	    // Manage step transitions and reset
	    #_step(forceReset := NOT #activate,
	           step := #step);
	    #_stepTracker.actual := #step.actual;
	END_REGION

	REGION Equipment Modules
	    REGION Vacuum: Commands
	        CASE #step.actual OF
	            VacHop_FlowThrough_Steps#RESET_STEP:
	                // Set vacuum to idle
	                #cmd_em_vacuum := _.EM_Vac.Vac_Cmd#IDLE;

	            VacHop_FlowThrough_Steps#INITIAL:
	                // Start vacuum or wait for idle
	                IF #em_vacuum_startVacuum_idle THEN
	                    #cmd_em_vacuum := _.EM_Vac.Vac_Cmd#IDLE;
	                ELSE
	                    #cmd_em_vacuum := _.EM_Vac.Vac_Cmd#START_VACUUM;
	                END_IF;
	            ELSE
	                // Maintain vacuum active
	                #cmd_em_vacuum := _.EM_Vac.Vac_Cmd#START_VACUUM;
	        END_CASE;

	    END_REGION

	    REGION Outlet Valve: Command
	        CASE #step.actual OF
	            VacHop_FlowThrough_Steps#RESET_STEP:
	                // Set outlet valve to idle
	                #cmd_em_outVlv := _.EM_outVlv.OutVlv_Cmd#IDLE;

	            VacHop_FlowThrough_Steps#INITIAL..VacHop_FlowThrough_Steps#CREATE_VACUUM:
	                // Open outlet valve or wait for close
	                IF NOT #em_outVlv_outletClose THEN
	                    #cmd_em_outVlv := _.EM_outVlv.OutVlv_Cmd#OPEN_OUTLET;

	                END_IF;
	            ELSE
	                // Maintain outlet valve open
	                #cmd_em_outVlv := _.EM_outVlv.OutVlv_Cmd#OPEN_OUTLET;

	        END_CASE;

	    END_REGION

	END_REGION

	REGION Control Modules: Commands
	    //********************************************************
	    // NA
	    //********************************************************

	END_REGION

	REGION Feedbacks
	    // na

	END_REGION

	REGION Status
	    // System idle when not activated
	    #status.idle := NOT #activate;

	    // System done when flowthrough complete
	    #status.done := NOT #status.idle AND #cm_inPosition AND #em_idleOrDone AND (#step.actual = VacHop_FlowThrough_Steps#READY);

	    //System busy during flowthrough sequence
	    #status.busy := NOT #status.idle AND NOT #status.done;

	END_REGION


END_FUNCTION_BLOCK
END_NAMESPACE

NAMESPACE EM_VacHop
TYPE VacHop_interface
{ Published := 'TRUE' }
VERSION : 0.1
   STRUCT
      cmd { ExternalAccessible := 'False'; ExternalVisible := 'False'; ExternalWritable := 'False'} : VacHop_Cmd;
      status { ExternalAccessible := 'False'; ExternalVisible := 'False'; ExternalWritable := 'False'; S7_SetPoint := 'False'} : _.LIB.Util_status;
      modesStatus { ExternalAccessible := 'False'; ExternalVisible := 'False'; ExternalWritable := 'False'; S7_SetPoint := 'False'} : VacHop_interface_modesStatus;
      feedbacks { ExternalAccessible := 'False'; ExternalVisible := 'False'; ExternalWritable := 'False'; S7_SetPoint := 'False'} : VacHop_interface_feedbacks;
   END_STRUCT;

END_TYPE
END_NAMESPACE

NAMESPACE EM_VacHop
FUNCTION_BLOCK EM_VacHop_evacuate
{ S7_Optimized_Access := 'TRUE' ; Published := 'TRUE' }
VERSION : 0.1
   VAR_INPUT
      enableStepTransition { ExternalAccessible := 'False'; ExternalVisible := 'False'; ExternalWritable := 'False'} : Bool := true;   // Enable Step Transition
      parameters { ExternalAccessible := 'False'; ExternalVisible := 'False'; ExternalWritable := 'False'} : VacHop_Evacuate_Params;
      activate { ExternalAccessible := 'False'; ExternalVisible := 'False'; ExternalWritable := 'False'} : Bool;
      cm_inPosition { ExternalAccessible := 'False'; ExternalVisible := 'False'; ExternalWritable := 'False'} : Bool;   // CM in position
      em_idleOrDone { ExternalAccessible := 'False'; ExternalVisible := 'False'; ExternalWritable := 'False'} : Bool;   // EM Idle or Done
      em_vacuum_startVacuum_idle { ExternalAccessible := 'False'; ExternalVisible := 'False'; ExternalWritable := 'False'} : Bool;   // EM Vacuum: Start Vacuum mode idle
      em_outVlv_outletClose { ExternalAccessible := 'False'; ExternalVisible := 'False'; ExternalWritable := 'False'} : Bool;   // EM_OutVlv: outlet valve is open
   END_VAR

   VAR_OUTPUT
      cmd_em_vacuum { ExternalAccessible := 'False'; ExternalVisible := 'False'; ExternalWritable := 'False'} : _.EM_Vac.Vac_Cmd;   // EM_Vacuum: Command
      cmd_em_outVlv { ExternalAccessible := 'False'; ExternalVisible := 'False'; ExternalWritable := 'False'} : _.EM_OutVlv.OutVlv_Cmd;   // EM_OutVlv: Command
   END_VAR

   VAR
      status { ExternalAccessible := 'False'; ExternalVisible := 'False'; ExternalWritable := 'False'; S7_SetPoint := 'False'} : _.LIB.Util_modeStatus;   // Mode status
      feedbacks { ExternalAccessible := 'False'; ExternalVisible := 'False'; ExternalWritable := 'False'; S7_SetPoint := 'False'} : VacHop_Evacuate_Feedbacks;   // Feedbacks
      step { ExternalAccessible := 'False'; ExternalVisible := 'False'; ExternalWritable := 'False'; S7_SetPoint := 'False'} : _.LIB.Util_Step;   // Step status
      _step { ExternalAccessible := 'False'; ExternalVisible := 'False'; ExternalWritable := 'False'; S7_SetPoint := 'False'} : _.LIB.Step;   // Step instance
      _stepTracker { ExternalAccessible := 'False'; ExternalVisible := 'False'; ExternalWritable := 'False'} : Struct
         actual { ExternalAccessible := 'False'; ExternalVisible := 'False'; ExternalWritable := 'False'} : VacHop_Evacuate_Steps;   // Current step
         next { ExternalAccessible := 'False'; ExternalVisible := 'False'; ExternalWritable := 'False'} : VacHop_Evacuate_Steps;   // Next step
      END_STRUCT;
   END_VAR


BEGIN
	REGION Header
	    //********************************************************
	    // EM_VacHop_evacuate Logic
	    // Description:
	    // - Manages the evacuation sequence for the vacuum hopper, closing the outlet and starting the vacuum system.
	    //********************************************************

	    REGION Revision History
	        (*
	        Author      Date        Change
	        GEA-VAR     2025-05-15  Initial version
	        *)
	    END_REGION
	END_REGION

	REGION Step
	    IF #activate THEN
	        CASE #step.actual OF
	                // Idle state, no sequence active
	            VacHop_Evacuate_Steps#INITIAL:
	                #_stepTracker.next := VacHop_Evacuate_Steps#CLOSE_OUTLET;

	                // Close outlet valve
	            VacHop_Evacuate_Steps#CLOSE_OUTLET:
	                #_stepTracker.next := VacHop_Evacuate_Steps#CREATE_VACUUM;

	                //  Start vacuum system
	            VacHop_Evacuate_Steps#CREATE_VACUUM:
	                #_stepTracker.next := VacHop_Evacuate_Steps#DONE;

	                //  Evacuation sequence complete
	            VacHop_Evacuate_Steps#DONE:
	                ;

	                // Handle invalid step
	            ELSE
	                // Reset to idle on invalid step
	                #step.actual := #_stepTracker.next := VacHop_Evacuate_Steps#INITIAL;
	        END_CASE;

	        // Advance step when module positioned
	        IF #enableStepTransition AND #cm_inPosition AND #em_idleOrDone THEN
	            #step.actual := #_stepTracker.next;
	        END_IF;

	    END_IF;

	    // Manage step transitions and reset
	    #_step(forceReset := NOT #activate,
	           step := #step);
	    #_stepTracker.actual := #step.actual;

	END_REGION

	REGION Equipment Modules
	    REGION Vacuum: Commands
	        CASE #step.actual OF
	            VacHop_Evacuate_Steps#RESET_STEP:
	                #cmd_em_vacuum := _.EM_Vac.Vac_Cmd#IDLE;

	            VacHop_Evacuate_Steps#INITIAL..VacHop_Evacuate_Steps#CLOSE_OUTLET:
	                IF #em_vacuum_startVacuum_idle THEN
	                    #cmd_em_vacuum := _.EM_Vac.Vac_Cmd#IDLE;
	                ELSE
	                    #cmd_em_vacuum := _.EM_Vac.Vac_Cmd#START_VACUUM;
	                END_IF;
	            ELSE
	                #cmd_em_vacuum := _.EM_Vac.Vac_Cmd#START_VACUUM;
	        END_CASE;

	    END_REGION

	    REGION Outlet Valve: Command
	        CASE #step.actual OF
	            VacHop_Evacuate_Steps#INITIAL..VacHop_Evacuate_Steps#CLOSE_OUTLET:
	                IF NOT #em_outVlv_outletClose THEN
	                    #cmd_em_outVlv := _.EM_outVlv.OutVlv_Cmd#CLOSE_OUTLET;
	                ELSE
	                    #cmd_em_outVlv := _.EM_outVlv.OutVlv_Cmd#IDLE;
	                END_IF;
	            ELSE
	                #cmd_em_outVlv := _.EM_outVlv.OutVlv_Cmd#IDLE;

	        END_CASE;

	    END_REGION

	END_REGION

	REGION Control Modules: Commands
	    //********************************************************
	    // NA
	    //********************************************************

	END_REGION

	REGION Feedbacks
	    // NA

	END_REGION

	REGION Status
	    // System idle when not activated
	    #status.idle := NOT #activate;

	    // System done when evacuation complete
	    #status.done := NOT #status.idle AND #cm_inPosition AND #em_idleOrDone AND (#step.actual = VacHop_Evacuate_Steps#DONE);

	    // System busy during evacuation sequence
	    #status.busy := NOT #status.idle AND NOT #status.done;

	END_REGION


END_FUNCTION_BLOCK
END_NAMESPACE

NAMESPACE EM_VacHop
FUNCTION_BLOCK EM_VacHop_openHopper
{ S7_Optimized_Access := 'TRUE' ; Published := 'TRUE' }
VERSION : 0.1
   VAR_INPUT
      enableStepTransition { ExternalAccessible := 'False'; ExternalVisible := 'False'; ExternalWritable := 'False'} : Bool := true;   // Enable Step Transition
      parameters { ExternalAccessible := 'False'; ExternalVisible := 'False'; ExternalWritable := 'False'} : VacHop_OpenHopper_Params;   // Open hopper parameters
      activate { ExternalAccessible := 'False'; ExternalVisible := 'False'; ExternalWritable := 'False'} : Bool;   // Activate open sequence
      cm_inPosition { ExternalAccessible := 'False'; ExternalVisible := 'False'; ExternalWritable := 'False'} : Bool;   // CM in position
      em_idleOrDone { ExternalAccessible := 'False'; ExternalVisible := 'False'; ExternalWritable := 'False'} : Bool;   // EM Idle or Done
      em_vacuum_idle { ExternalAccessible := 'False'; ExternalVisible := 'False'; ExternalWritable := 'False'} : Bool;   // EM Vacuum:  idle
      em_outVlv_outletClose { ExternalAccessible := 'False'; ExternalVisible := 'False'; ExternalWritable := 'False'} : Bool;   // EM_OutVlv outlet valve closed
   END_VAR

   VAR_OUTPUT
      cmd_em_vacuum { ExternalAccessible := 'False'; ExternalVisible := 'False'; ExternalWritable := 'False'} : _.EM_Vac.Vac_Cmd;   // EM_Vacuum: Command
      cmd_em_outVlv { ExternalAccessible := 'False'; ExternalVisible := 'False'; ExternalWritable := 'False'} : _.EM_OutVlv.OutVlv_Cmd;   // EM_Hopper: Command
   END_VAR

   VAR
      status { ExternalAccessible := 'False'; ExternalVisible := 'False'; ExternalWritable := 'False'; S7_SetPoint := 'False'} : _.LIB.Util_modeStatus;   // Mode status
      feedbacks { ExternalAccessible := 'False'; ExternalVisible := 'False'; ExternalWritable := 'False'; S7_SetPoint := 'False'} : VacHop_OpenHopper_Feedbacks;   // Feedbacks
      step { ExternalAccessible := 'False'; ExternalVisible := 'False'; ExternalWritable := 'False'; S7_SetPoint := 'False'} : _.LIB.Util_Step;   // Step status
      _step { ExternalAccessible := 'False'; ExternalVisible := 'False'; ExternalWritable := 'False'; S7_SetPoint := 'False'} : _.LIB.Step;   // Step instance
      _stepTracker { ExternalAccessible := 'False'; ExternalVisible := 'False'; ExternalWritable := 'False'} : Struct
         actual { ExternalAccessible := 'False'; ExternalVisible := 'False'; ExternalWritable := 'False'} : VacHop_OpenHopper_Steps;   // Current step
         next { ExternalAccessible := 'False'; ExternalVisible := 'False'; ExternalWritable := 'False'} : VacHop_OpenHopper_Steps;   // Next step
      END_STRUCT;
   END_VAR


BEGIN
	REGION Header
	    //********************************************************
	    // EM_VacHop_openHopper Logic
	    // Description:
	    // - Manages the hopper outlet opening sequence for the vacuum hopper, stopping vacuum and opening the outlet valve.
	    //********************************************************

	    REGION Revision History
	        (*
	        Author      Date        Change
	        GEA-VAR     2025-05-15  Initial version
	        *)
	    END_REGION
	END_REGION

	REGION Step
	    IF #activate THEN
	        CASE #step.actual OF
	                // Idle state, no sequence active
	            VacHop_OpenHopper_Steps#INITIAL:
	                #_stepTracker.next := VacHop_OpenHopper_Steps#STOP_VACUUM;

	                // Stop vacuum system
	            VacHop_OpenHopper_Steps#STOP_VACUUM:
	                #_stepTracker.next := VacHop_OpenHopper_Steps#OPEN_OUTLET;

	                //  Open outlet valve
	            VacHop_OpenHopper_Steps#OPEN_OUTLET:
	                #_stepTracker.next := VacHop_OpenHopper_Steps#DONE;

	                //  Outlet valve opened, sequence complete
	            VacHop_OpenHopper_Steps#DONE:
	                ;

	                // Handle invalid step
	            ELSE
	                // Reset to idle on invalid step
	                #step.actual := #_stepTracker.next := VacHop_OpenHopper_Steps#INITIAL;
	        END_CASE;

	        // Advance step when module positioned
	        IF #enableStepTransition AND #cm_inPosition AND #em_idleOrDone THEN
	            #step.actual := #_stepTracker.next;
	        END_IF;

	    END_IF;

	    // Manage step transitions and reset
	    #_step(forceReset := NOT #activate,
	           step := #step);
	    #_stepTracker.actual := #step.actual;

	END_REGION

	REGION Control/Equipment Modules and Modes: Commands

	    REGION Vacuum: Commands
	        CASE #step.actual OF
	            VacHop_OpenHopper_Steps#INITIAL..VacHop_OpenHopper_Steps#STOP_VACUUM:
	                IF #em_vacuum_idle THEN
	                    #cmd_em_vacuum := _.EM_Vac.Vac_Cmd#IDLE;
	                ELSE
	                    #cmd_em_vacuum := _.EM_Vac.Vac_Cmd#STOP_VACUUM;
	                END_IF;
	            ELSE
	                #cmd_em_vacuum := _.EM_Vac.Vac_Cmd#IDLE;
	        END_CASE;

	    END_REGION

	    REGION Outlet Valve: Command
	        CASE #step.actual OF
	            VacHop_OpenHopper_Steps#RESET_STEP:
	                #cmd_em_outVlv := _.EM_outVlv.OutVlv_Cmd#IDLE;

	            VacHop_OpenHopper_Steps#INITIAL..VacHop_OpenHopper_Steps#STOP_VACUUM:
	                IF NOT #em_outVlv_outletClose THEN
	                    #cmd_em_outVlv := _.EM_outVlv.OutVlv_Cmd#OPEN_OUTLET;
	                ELSE
	                    #cmd_em_outVlv := _.EM_outVlv.OutVlv_Cmd#IDLE;
	                END_IF;
	            ELSE
	                #cmd_em_outVlv := _.EM_outVlv.OutVlv_Cmd#OPEN_OUTLET;
	        END_CASE;

	    END_REGION

	END_REGION

	REGION Control Modules: Commands
	    //********************************************************
	    // NA
	    //********************************************************

	END_REGION

	REGION Feedbacks
	    // NA

	END_REGION

	REGION Status
	    // System idle when not activated
	    #status.idle := NOT #activate;

	    // System done when hopper opened
	    #status.done := (NOT #status.idle) AND #cm_inPosition AND #em_idleOrDone AND (#step.actual = VacHop_OpenHopper_Steps#DONE);

	    // System busy during open sequence
	    #status.busy := NOT #status.idle AND NOT #status.done;

	END_REGION


END_FUNCTION_BLOCK
END_NAMESPACE

NAMESPACE EM_VacHop
FUNCTION_BLOCK EM_VacHop_vent
{ S7_Optimized_Access := 'TRUE' ; Published := 'TRUE' }
VERSION : 0.1
   VAR_INPUT
      enableStepTransition { ExternalAccessible := 'False'; ExternalVisible := 'False'; ExternalWritable := 'False'} : Bool := true;   // Enable Step Transition
      parameters { ExternalAccessible := 'False'; ExternalVisible := 'False'; ExternalWritable := 'False'} : VacHop_Vent_Params;   // Vent parameters
      activate { ExternalAccessible := 'False'; ExternalVisible := 'False'; ExternalWritable := 'False'} : Bool;   // Activate vent sequence
      cm_inPosition { ExternalAccessible := 'False'; ExternalVisible := 'False'; ExternalWritable := 'False'} : Bool;   // CM in position
      em_idleOrDone { ExternalAccessible := 'False'; ExternalVisible := 'False'; ExternalWritable := 'False'} : Bool;   // EM Idle or Done
      em_vacuum_idle { ExternalAccessible := 'False'; ExternalVisible := 'False'; ExternalWritable := 'False'} : Bool;   // EM Vacuum:  idle
      em_outVlv_outletClose { ExternalAccessible := 'False'; ExternalVisible := 'False'; ExternalWritable := 'False'} : Bool;   // EM_outVlv: outlet valve is closed
   END_VAR

   VAR_OUTPUT
      cmd_em_vacuum { ExternalAccessible := 'False'; ExternalVisible := 'False'; ExternalWritable := 'False'} : _.EM_Vac.Vac_Cmd;   // EM_Vacuum: Command
      cmd_em_outVlv { ExternalAccessible := 'False'; ExternalVisible := 'False'; ExternalWritable := 'False'} : _.EM_OutVlv.OutVlv_Cmd;   // EM_outVlv: Command
      cmd_ventVlvOpen { ExternalAccessible := 'False'; ExternalVisible := 'False'; ExternalWritable := 'False'} : Bool;   // Command vent valve open
   END_VAR

   VAR
      status { ExternalAccessible := 'False'; ExternalVisible := 'False'; ExternalWritable := 'False'; S7_SetPoint := 'False'} : _.LIB.Util_modeStatus;   // Mode status
      feedbacks { ExternalAccessible := 'False'; ExternalVisible := 'False'; ExternalWritable := 'False'; S7_SetPoint := 'False'} : VacHop_Vent_Feedbacks;   // Feedbacks
      step { ExternalAccessible := 'False'; ExternalVisible := 'False'; ExternalWritable := 'False'; S7_SetPoint := 'False'} : _.LIB.Util_Step;   // Step status
      _step { ExternalAccessible := 'False'; ExternalVisible := 'False'; ExternalWritable := 'False'; S7_SetPoint := 'False'} : _.LIB.Step;   // Step instance
      _stepTracker { ExternalAccessible := 'False'; ExternalVisible := 'False'; ExternalWritable := 'False'} : Struct
         actual { ExternalAccessible := 'False'; ExternalVisible := 'False'; ExternalWritable := 'False'} : VacHop_Vent_Steps;   // Current step
         next { ExternalAccessible := 'False'; ExternalVisible := 'False'; ExternalWritable := 'False'} : VacHop_Vent_Steps;   // Next step
      END_STRUCT;
   END_VAR


BEGIN
	REGION Header
	    //********************************************************
	    // EM_VacHop_vent Logic
	    // Description:
	    // - Manages the vent sequence for the vacuum hopper, stopping vacuum, closing outlet, and cycling the vent valve.
	    //********************************************************

	    REGION Revision History
	        (*
	        Author      Date        Change
	        GEA-VAR     2025-05-15  Initial version
	        *)
	    END_REGION
	END_REGION

	REGION Step
	    IF #activate THEN
	        CASE #step.actual OF
	                // Idle state, no sequence active
	            VacHop_Vent_Steps#INITIAL:
	                #_stepTracker.next := VacHop_Vent_Steps#STOP_VACUUM_AND_CLOSE_OUTLET;

	                // Stop vacuum and close outlet valve
	            VacHop_Vent_Steps#STOP_VACUUM_AND_CLOSE_OUTLET:
	                #_stepTracker.next := VacHop_Vent_Steps#OPEN_VENT_VALVE;

	                //  Open vent valve
	            VacHop_Vent_Steps#OPEN_VENT_VALVE:
	                #_stepTracker.next := VacHop_Vent_Steps#VENT_DELAY_ACTIVE;

	                //  Delay for venting
	            VacHop_Vent_Steps#VENT_DELAY_ACTIVE:
	                IF _.LIB.IsTimerExceeded(actualTimer:=#step.actualTimer, limit:=#parameters.ventTime) THEN
	                    #_stepTracker.next := VacHop_Vent_Steps#CLOSE_VENT_VALVE;
	                END_IF;

	                // Close vent valve
	            VacHop_Vent_Steps#CLOSE_VENT_VALVE:
	                #_stepTracker.next := VacHop_Vent_Steps#DONE;

	                // Vent sequence complete
	            VacHop_Vent_Steps#DONE:
	                ;

	                // Handle invalid step
	            ELSE
	                // Reset to idle on invalid step
	                #step.actual := #_stepTracker.next := VacHop_Vent_Steps#INITIAL;
	        END_CASE;

	        // Advance step when module positioned
	        IF #enableStepTransition AND #cm_inPosition AND #em_idleOrDone THEN
	            #step.actual := #_stepTracker.next;
	        END_IF;

	    END_IF;

	    // Manage step transitions and reset
	    #_step(forceReset:=NOT #activate,
	           step := #step);
	    #_stepTracker.actual := #step.actual;
	END_REGION

	REGION Actions
	    // NA

	END_REGION

	REGION Control/Equipment Modules and Modes: Commands
	    REGION Vacuum: Commands
	        CASE #step.actual OF
	            VacHop_Vent_Steps#INITIAL..VacHop_Vent_Steps#STOP_VACUUM_AND_CLOSE_OUTLET:
	                IF #em_vacuum_idle THEN
	                    #cmd_em_vacuum := _.EM_Vac.Vac_Cmd#IDLE;
	                ELSE
	                    #cmd_em_vacuum := _.EM_Vac.Vac_Cmd#STOP_VACUUM;
	                END_IF;
	            ELSE
	                #cmd_em_vacuum := _.EM_Vac.Vac_Cmd#IDLE;
	        END_CASE;

	    END_REGION

	    REGION Vacuum valve: Command
	        CASE #step.actual OF
	            VacHop_Vent_Steps#INITIAL..VacHop_Vent_Steps#STOP_VACUUM_AND_CLOSE_OUTLET:
	                IF NOT #em_outVlv_outletClose THEN
	                    #cmd_em_outVlv := _.EM_outVlv.OutVlv_Cmd#CLOSE_OUTLET;
	                ELSE
	                    #cmd_em_outVlv := _.EM_outVlv.OutVlv_Cmd#IDLE;
	                END_IF;
	            ELSE
	                #cmd_em_outVlv := _.EM_outVlv.OutVlv_Cmd#IDLE;
	        END_CASE;

	    END_REGION

	END_REGION

	REGION Control Modules: Commands
	    //********************************************************
	    // Vent Valve
	    //********************************************************
	    #cmd_ventVlvOpen := #activate AND (NOT (#step.actual = VacHop_Vent_Steps#CLOSE_VENT_VALVE)) AND (NOT ((#step.actual = VacHop_Vent_Steps#DONE)));


	END_REGION

	REGION #feedbacks
	    // Update feedback statuses
	    #feedbacks.venting := (#step.actual = VacHop_Vent_Steps#OPEN_VENT_VALVE) OR (#step.actual = VacHop_Vent_Steps#VENT_DELAY_ACTIVE);

	END_REGION

	REGION Status
	    // System idle when not activated
	    #status.idle := NOT #activate;

	    // System done when vent complete
	    #status.done := (NOT #status.idle) AND #cm_inPosition AND #em_idleOrDone AND (#step.actual = VacHop_Vent_Steps#DONE);

	    // System busy during vent sequence
	    #status.busy := NOT #status.idle AND NOT #status.done;

	END_REGION


END_FUNCTION_BLOCK
END_NAMESPACE

NAMESPACE EM_OutVlv
FUNCTION_BLOCK EM_OutVlv
{ S7_Optimized_Access := 'TRUE' ; Published := 'TRUE' }
VERSION : 0.1
   VAR_INPUT
      enableStepTransition { ExternalAccessible := 'False'; ExternalVisible := 'False'; ExternalWritable := 'False'} : Bool := True;   // Enable step transition
      outletValveInputs { ExternalAccessible := 'False'; ExternalVisible := 'False'; ExternalWritable := 'False'} : OutVlv_inputs;   // EM inputs
   END_VAR

   VAR_OUTPUT
      cm_inPosition { ExternalAccessible := 'False'; ExternalVisible := 'False'; ExternalWritable := 'False'} : Bool;   // CM in position
      cmd_outletVlvOpen { ExternalAccessible := 'False'; ExternalVisible := 'False'; ExternalWritable := 'False'} : Bool;   // Command: outlet valve open
   END_VAR

   VAR
      interface { ExternalAccessible := 'False'; ExternalVisible := 'False'; ExternalWritable := 'False'; S7_SetPoint := 'False'} : OutVlv_interface;
      parameters : OutVlv_parameters;
      _initialize { ExternalAccessible := 'False'; ExternalVisible := 'False'; ExternalWritable := 'False'; S7_SetPoint := 'False'} : EM_OutVlv_initialize;
      _purge { ExternalAccessible := 'False'; ExternalVisible := 'False'; ExternalWritable := 'False'; S7_SetPoint := 'False'} : EM_OutVlv_purge;
      _discharge { ExternalAccessible := 'False'; ExternalVisible := 'False'; ExternalWritable := 'False'; S7_SetPoint := 'False'} : EM_OutVlv_discharge;
      _holdPosition { ExternalAccessible := 'False'; ExternalVisible := 'False'; ExternalWritable := 'False'; S7_SetPoint := 'False'} : EM_OutVlv_holdPosition;
      _openOutlet { ExternalAccessible := 'False'; ExternalVisible := 'False'; ExternalWritable := 'False'; S7_SetPoint := 'False'} : EM_OutVlv_openOutlet;
      _closeOutlet { ExternalAccessible := 'False'; ExternalVisible := 'False'; ExternalWritable := 'False'; S7_SetPoint := 'False'} : EM_OutVlv_closeOutlet;
      _outputs { ExternalAccessible := 'False'; ExternalVisible := 'False'; ExternalWritable := 'False'} : Struct
         cmd_outletVlvOpen { ExternalAccessible := 'False'; ExternalVisible := 'False'; ExternalWritable := 'False'} : Bool;
      END_STRUCT;
   END_VAR

   VAR_TEMP
      temp_mode_idle_or_done : Bool;
   END_VAR


BEGIN
	REGION Header
	    //********************************************************
	    // EM_OutVlv Logic
	    // Description:
	    // - Main controller for the outlet valvce system.
	    //********************************************************

	    REGION Revision History
	        (*
	            Author      Date        Change
	            GEA-VAR     15MAY25     Initial version
	        *)
	    END_REGION

	END_REGION

	REGION Check CM/EM(mode) in position
	    // Set control module position status
	    #cm_inPosition :=
	        (#_outputs.cmd_outletVlvOpen AND #outletValveInputs.outletVlv_isOpen) OR
	        ((NOT #_outputs.cmd_outletVlvOpen) AND #outletValveInputs.outletVlv_isClosed);

	    #temp_mode_idle_or_done :=
	        (#_openOutlet.status.idle OR #_openOutlet.status.done) AND
	        (#_closeOutlet.status.idle OR #_closeOutlet.status.done);

	END_REGION

	REGION Initialize
	    // Run initialization sequence
	    #_initialize(enableStepTransition:=#enableStepTransition,
	                 activate:=(#interface.cmd = OutVlv_Cmd#INITIALIZE),
	                 cm_inPosition:=#cm_inPosition,
	                 mode_idleOrDone:=#temp_mode_idle_or_done);

	END_REGION

	REGION Purge
	    REGION Parameters
	        // Configure parameters for the purge count
	        #_purge.parameters.startDelay := #parameters.fixed.purgeStartDelay;
	        #_purge.parameters.count := #parameters.fixed.purgeCount;
	        #_purge.parameters.outletVlvOpenDelay := #parameters.fixed.purgeOutletVlvOpenDelay;
	        #_purge.parameters.outletVlvCloseDelay := #parameters.fixed.purgeOutletVlvCloseDelay;

	    END_REGION

	    // Activate Purge sequence on command
	    #_purge(enableStepTransition:=#enableStepTransition,
	            activate := (#interface.cmd = OutVlv_Cmd#PURGE),
	            cm_inPosition:=#cm_inPosition,
	            mode_idleOrDone:=#temp_mode_idle_or_done,
	            outletVlv_isOpen:=#outletValveInputs.outletVlv_isOpen);
	END_REGION

	REGION Discharge
	    // Configure parameters for the discharge mode
	    REGION Parameters
	        #_discharge.parameters.dischargeTime := #parameters.variable.dischargeTime;

	    END_REGION

	    // Activate Purge sequence on command
	    #_discharge(enableStepTransition:=#enableStepTransition,
	                activate := (#interface.cmd = OutVlv_Cmd#DISCHARGE),
	                cm_inPosition:=#cm_inPosition,
	                mode_idleOrDone:=#temp_mode_idle_or_done);
	END_REGION

	REGION Hold Position
	    // Configure parameters for the Hold Position mode
	    REGION Parameters
	        #_holdPosition.parameters.na := FALSE;

	    END_REGION

	    // Activate Hold Position sequence on command
	    #_holdPosition(enableStepTransition:=#enableStepTransition,
	                   activate := (#interface.cmd = OutVlv_Cmd#HOLD_POSITION),
	                   cm_inPosition := #cm_inPosition,
	                   mode_idleOrDone := #temp_mode_idle_or_done,
	                   outletVlv_isClosed:=#outletValveInputs.outletVlv_isClosed);
	END_REGION

	REGION Open Outlet
	    // Configure parameters for the open outlet delay
	    REGION Parameters
	        IF #_purge.cmd_modeOpenOutlet THEN
	            #_openOutlet.parameters.vlvOpenDelay := #_purge.parameters.outletVlvOpenDelay;
	        ELSE
	            #_openOutlet.parameters.vlvOpenDelay := #parameters.fixed.outletVlvOpenDelay;
	        END_IF;

	    END_REGION

	    // Activate Open Outlet sequence when commanded or required by initialization, purge, discharge or holdPosition
	    #_openOutlet(enableStepTransition:=#enableStepTransition,
	                 activate := (#interface.cmd = OutVlv_Cmd#OPEN_OUTLET) OR #_initialize.cmd_modeOpenOutlet OR #_purge.cmd_modeOpenOutlet OR #_discharge.cmd_modeOpenOutlet OR #_holdPosition.cmd_modeOpenOutlet,
	                 cm_inPosition:=#cm_inPosition,
	                 outletVlv_isOpen:=#outletValveInputs.outletVlv_isOpen);

	END_REGION

	REGION Close Outlet
	    // Configure parameters for the close outlet delay
	    REGION Parameters
	        IF #_purge.cmd_modeCloseOutlet THEN
	            #_closeOutlet.parameters.vlvCloseDelay := #_purge.parameters.outletVlvCloseDelay;
	        ELSE
	            #_closeOutlet.parameters.vlvCloseDelay := #parameters.fixed.outletVlvCloseDelay;
	        END_IF;

	    END_REGION

	    // Activate Close Outlet sequence when commanded or required by initialization, purge, discharge or holdPosition
	    #_closeOutlet(enableStepTransition:=#enableStepTransition,
	                  activate := (#interface.cmd = OutVlv_Cmd#CLOSE_OUTLET) OR #_initialize.cmd_modeCloseOutlet OR #_purge.cmd_modeCloseOutlet OR #_discharge.cmd_modeCloseOutlet OR #_holdPosition.cmd_modeCloseOutlet,
	                  cm_inPosition:=#cm_inPosition,
	                  outletVlv_isOpen := #outletValveInputs.outletVlv_isOpen,
	                  outletVlv_isClosed := #outletValveInputs.outletVlv_isClosed);
	END_REGION


	REGION Outputs
	    // Combine valve commands from outlet sequences
	    #cmd_outletVlvOpen := #_outputs.cmd_outletVlvOpen := #_openOutlet.cmd_outletVlvOpen OR #_closeOutlet.cmd_outletVlvOpen;

	END_REGION

	REGION Feedbacks
	    // Update mode feedbacks
	    #interface.feedbacks.outletOpen := #outletValveInputs.outletVlv_isOpen;
	    #interface.feedbacks.openingOutlet := (NOT #outletValveInputs.outletVlv_isOpen) AND #cmd_outletVlvOpen;
	    #interface.feedbacks.outletClose := #outletValveInputs.outletVlv_isClosed;
	    #interface.feedbacks.closingOutlet := (NOT #outletValveInputs.outletVlv_isClosed) AND (#interface.cmd <> OutVlv_Cmd#IDLE) AND  (NOT #cmd_outletVlvOpen);
	    #interface.feedbacks.held := #_holdPosition.feedbacks.held;

	    REGION Modes
	        #interface.feedbacks.modes.initialize := #_initialize.feedbacks;
	        #interface.feedbacks.modes.openOutlet := #_openOutlet.feedbacks;
	        #interface.feedbacks.modes.closeOutlet := #_closeOutlet.feedbacks;
	        #interface.feedbacks.modes.purge := #_purge.feedbacks;
	        #interface.feedbacks.modes.discharge := #_discharge.feedbacks;
	        #interface.feedbacks.modes.holdPosition := #_holdPosition.feedbacks;

	    END_REGION

	END_REGION


	REGION Check CM/EM(mode) in position
	    // Set control module position status
	    #cm_inPosition :=
	        (#_outputs.cmd_outletVlvOpen AND #outletValveInputs.outletVlv_isOpen) OR
	        ((NOT #_outputs.cmd_outletVlvOpen) AND #outletValveInputs.outletVlv_isClosed);

	    // Check if modes are idle or done
	    #temp_mode_idle_or_done :=
	        (#_openOutlet.status.idle OR #_openOutlet.status.done) AND
	        (#_closeOutlet.status.idle OR #_closeOutlet.status.done);

	END_REGION

	REGION Status
	    #interface.status.done := #_initialize.status.done OR #_purge.status.done OR #_discharge.status.done OR #_holdPosition.status.done OR
	    ((NOT (#_initialize.status.busy OR #_purge.status.busy OR #_discharge.status.busy OR #_holdPosition.status.busy)) AND (#_openOutlet.status.done OR #_closeOutlet.status.done));
	    #interface.status.busy := #_initialize.status.busy OR #_openOutlet.status.busy OR #_closeOutlet.status.busy OR #_purge.status.busy OR #_discharge.status.busy;
	    #interface.status.idle := NOT (#interface.status.busy OR #interface.status.done);
	    #interface.status.stopAlmActive := _.EM.TODO.alm;
	    #interface.status.abortAlmActive := _.EM.TODO.alm;

	    // Modes
	    #interface.modesStatus.initialize := #_initialize.status;
	    #interface.modesStatus.openOutlet := #_openOutlet.status;
	    #interface.modesStatus.closeOutlet := #_closeOutlet.status;
	    #interface.modesStatus.purge := #_purge.status;
	    #interface.modesStatus.discharge := #_discharge.status;
	    #interface.modesStatus.holdPosition := #_holdPosition.status;

	END_REGION

END_FUNCTION_BLOCK
END_NAMESPACE

NAMESPACE EM_VacHop
FUNCTION_BLOCK EM_VacHop_discharge
{ S7_Optimized_Access := 'TRUE' ; Published := 'TRUE' }
VERSION : 0.1
   VAR_INPUT
      enableStepTransition { ExternalAccessible := 'False'; ExternalVisible := 'False'; ExternalWritable := 'False'} : Bool := true;   // Enable Step Transition
      parameters { ExternalAccessible := 'False'; ExternalVisible := 'False'; ExternalWritable := 'False'} : VacHop_Discharge_Params;   // Discharge parameters
      activate { ExternalAccessible := 'False'; ExternalVisible := 'False'; ExternalWritable := 'False'} : Bool;   // Activate discharge sequence
      cm_inPosition { ExternalAccessible := 'False'; ExternalVisible := 'False'; ExternalWritable := 'False'} : Bool;   // CM in position
      em_idleOrDone { ExternalAccessible := 'False'; ExternalVisible := 'False'; ExternalWritable := 'False'} : Bool;   // EM Idle or Done
      em_vacuum_idle { ExternalAccessible := 'False'; ExternalVisible := 'False'; ExternalWritable := 'False'} : Bool;   // EM vacuum idle
      em_outVlv_outletClose { ExternalAccessible := 'False'; ExternalVisible := 'False'; ExternalWritable := 'False'} : Bool;   // EM_OutVlv: outlet valve is closed
   END_VAR

   VAR_OUTPUT
      cmd_em_vacuum { ExternalAccessible := 'False'; ExternalVisible := 'False'; ExternalWritable := 'False'} : _.EM_Vac.Vac_Cmd;   // EM_Vac command
      cmd_em_outVlv { ExternalAccessible := 'False'; ExternalVisible := 'False'; ExternalWritable := 'False'} : _.EM_OutVlv.OutVlv_Cmd;   // EM_OutVlv command
   END_VAR

   VAR
      status { ExternalAccessible := 'False'; ExternalVisible := 'False'; ExternalWritable := 'False'; S7_SetPoint := 'False'} : _.LIB.Util_modeStatus;   // Mode status
      feedbacks { ExternalAccessible := 'False'; ExternalVisible := 'False'; ExternalWritable := 'False'; S7_SetPoint := 'False'} : VacHop_Discharge_Feedbacks;   // Feedbacks
      step { ExternalAccessible := 'False'; ExternalVisible := 'False'; ExternalWritable := 'False'; S7_SetPoint := 'False'} : _.LIB.Util_Step;   // Step status
      _step { ExternalAccessible := 'False'; ExternalVisible := 'False'; ExternalWritable := 'False'; S7_SetPoint := 'False'} : _.LIB.Step;   // Step instance
      _stepTracker { ExternalAccessible := 'False'; ExternalVisible := 'False'; ExternalWritable := 'False'} : Struct
         actual { ExternalAccessible := 'False'; ExternalVisible := 'False'; ExternalWritable := 'False'} : VacHop_Discharge_Steps;   // Current step
         next { ExternalAccessible := 'False'; ExternalVisible := 'False'; ExternalWritable := 'False'} : VacHop_Discharge_Steps;   // Next step
      END_STRUCT;
   END_VAR


BEGIN
	REGION Header
	    //********************************************************
	    // EM_VacHop_discharge Logic
	    // Description:
	    // - Manages the discharge sequence for the vacuum hopper, stopping vacuum and opening the outlet valve.
	    //********************************************************

	    REGION Revision History
	        (*
	        Author      Date        Change
	        GEA-VAR     2025-05-15  Initial version
	        *)
	    END_REGION
	END_REGION

	REGION Step
	    IF #activate THEN
	        CASE #step.actual OF
	                // Idle state, no sequence active
	            VacHop_Discharge_Steps#INITIAL:
	                #_stepTracker.next := VacHop_Discharge_Steps#STOP_VACUUM;

	                // Stop vacuum system
	            VacHop_Discharge_Steps#STOP_VACUUM:
	                #_stepTracker.next := VacHop_Discharge_Steps#DISCHARGE;

	                // Discharge product
	            VacHop_Discharge_Steps#DISCHARGE:
	                #_stepTracker.next := VacHop_Discharge_Steps#DONE;

	                // Discharge sequence complete
	            VacHop_Discharge_Steps#DONE:
	                ;

	                // Handle invalid step
	            ELSE
	                // Reset to idle on invalid step
	                #step.actual := #_stepTracker.next := VacHop_Discharge_Steps#INITIAL;
	        END_CASE;

	        // Advance step when module positioned
	        IF #enableStepTransition AND  #cm_inPosition AND #em_idleOrDone THEN
	            #step.actual := #_stepTracker.next;
	        END_IF;

	    END_IF;

	    // Manage step transitions and reset
	    #_step(forceReset:=NOT #activate,
	           step := #step);
	    #_stepTracker.actual := #step.actual;
	END_REGION

	REGION Actions
	    // NA

	END_REGION

	REGION Equipment Modules
	    REGION Vacuum: Commands
	        CASE #step.actual OF
	            VacHop_Discharge_Steps#INITIAL..VacHop_Discharge_Steps#STOP_VACUUM:
	                // Stop vacuum or wait for idle
	                IF #em_vacuum_idle THEN
	                    #cmd_em_vacuum := _.EM_Vac.Vac_Cmd#IDLE;
	                ELSE
	                    #cmd_em_vacuum := _.EM_Vac.Vac_Cmd#STOP_VACUUM;
	                END_IF;
	            ELSE
	                // Maintain vacuum idle
	                #cmd_em_vacuum := _.EM_Vac.Vac_Cmd#IDLE;
	        END_CASE;

	    END_REGION

	    REGION Outlet Valve: Command
	        CASE #step.actual OF
	            VacHop_Discharge_Steps#INITIAL..VacHop_Discharge_Steps#STOP_VACUUM:
	                // Open outlet valve or wait for close
	                IF NOT #em_outVlv_outletClose THEN
	                    #cmd_em_outVlv := _.EM_outVlv.OutVlv_Cmd#OPEN_OUTLET;
	                ELSE
	                    #cmd_em_outVlv := _.EM_outVlv.OutVlv_Cmd#IDLE;

	                END_IF;

	            VacHop_Discharge_Steps#DISCHARGE:
	                // Discharge outlet valve
	                #cmd_em_outVlv := _.EM_outVlv.OutVlv_Cmd#DISCHARGE;

	            ELSE
	                #cmd_em_outVlv := _.EM_outVlv.OutVlv_Cmd#IDLE;

	        END_CASE;

	    END_REGION

	END_REGION

	REGION Control Modules: Commands
	    //********************************************************
	    // NA
	    //********************************************************

	END_REGION


	REGION Feedbacks
	    // Update feedback statuses
	    #feedbacks.discharging := (#step.actual = VacHop_Discharge_Steps#DISCHARGE);

	END_REGION

	//********************************************************
	// Region: #status Handling
	// Provides system status updates
	//********************************************************
	REGION Status
	    // System idle when not activated
	    #status.idle := NOT #activate;

	    // System done when discharge complete
	    #status.done := NOT #status.idle AND #cm_inPosition AND #em_idleOrDone AND (#step.actual = VacHop_Discharge_Steps#DONE);

	    // System busy during discharge sequence
	    #status.busy := NOT #status.idle AND NOT #status.done;

	END_REGION


END_FUNCTION_BLOCK
END_NAMESPACE

NAMESPACE EM_VacHop
FUNCTION_BLOCK EM_VacHop_initialize
{ S7_Optimized_Access := 'TRUE' ; Published := 'TRUE' }
VERSION : 0.1
   VAR_INPUT
      enableStepTransition { ExternalAccessible := 'False'; ExternalVisible := 'False'; ExternalWritable := 'False'} : Bool := true;   // Enable step transition
      activate { ExternalAccessible := 'False'; ExternalVisible := 'False'; ExternalWritable := 'False'} : Bool;   // Activate initialize sequence
      cm_inPosition { ExternalAccessible := 'False'; ExternalVisible := 'False'; ExternalWritable := 'False'} : Bool;   // CM/EM in position
      mode_idleOrDone { ExternalAccessible := 'False'; ExternalVisible := 'False'; ExternalWritable := 'False'} : Bool;   // Mode idle or done
   END_VAR

   VAR_OUTPUT
      cmd_em_vacuum { ExternalAccessible := 'False'; ExternalVisible := 'False'; ExternalWritable := 'False'} : _.EM_Vac.Vac_Cmd;   // EM_Vac command
      cmd_em_outVlv { ExternalAccessible := 'False'; ExternalVisible := 'False'; ExternalWritable := 'False'} : _.EM_OutVlv.OutVlv_Cmd;   // EM_OutVlv command
      cmd_modeVent { ExternalAccessible := 'False'; ExternalVisible := 'False'; ExternalWritable := 'False'} : Bool;   // Command vent mode
   END_VAR

   VAR
      status { ExternalAccessible := 'False'; ExternalVisible := 'False'; ExternalWritable := 'False'; S7_SetPoint := 'False'} : _.LIB.Util_modeStatus;   // Mode status
      feedbacks { ExternalAccessible := 'False'; ExternalVisible := 'False'; ExternalWritable := 'False'; S7_SetPoint := 'False'} : VacHop_Initialize_Feedbacks;   // Feedbacks
      step { ExternalAccessible := 'False'; ExternalVisible := 'False'; ExternalWritable := 'False'; S7_SetPoint := 'False'} : _.LIB.Util_Step;   // Step status
      _step { ExternalAccessible := 'False'; ExternalVisible := 'False'; ExternalWritable := 'False'; S7_SetPoint := 'False'} : _.LIB.Step;   // Step instance
      _stepTracker { ExternalAccessible := 'False'; ExternalVisible := 'False'; ExternalWritable := 'False'} : Struct
         actual { ExternalAccessible := 'False'; ExternalVisible := 'False'; ExternalWritable := 'False'} : VacHop_Initialize_Steps;   // Current step
         next { ExternalAccessible := 'False'; ExternalVisible := 'False'; ExternalWritable := 'False'} : VacHop_Initialize_Steps;   // Next step
      END_STRUCT;
   END_VAR


BEGIN
	REGION Header
	    //********************************************************
	    // EM_VacHop_initialize Logic
	    // Description:
	    // - Manages the initialization sequence for the vacuum hopper, initializing vacuum and outlet valve, then venting.
	    //********************************************************

	    REGION Revision History
	        (*
	        Author      Date        Change
	        GEA-VAR     2025-05-15  Initial version
	        *)
	    END_REGION
	END_REGION

	REGION Step
	    IF #activate THEN
	        CASE #step.actual OF
	                // Idle state, no sequence active
	            VacHop_Initialize_Steps#INITIAL:
	                #_stepTracker.next := VacHop_Initialize_Steps#INITIALIZE_VACUUM;

	                // Initialize vacuum
	            VacHop_Initialize_Steps#INITIALIZE_VACUUM:
	                #_stepTracker.next := VacHop_Initialize_Steps#INITIALIZE_HOPPER;

	                // Initialize hopper
	            VacHop_Initialize_Steps#INITIALIZE_HOPPER:
	                #_stepTracker.next := VacHop_Initialize_Steps#VENT;

	                // Vent
	            VacHop_Initialize_Steps#VENT:
	                #_stepTracker.next := VacHop_Initialize_Steps#INITIALIZED;

	                //  Initialization complete
	            VacHop_Initialize_Steps#INITIALIZED:
	                ;

	                // Handle invalid step
	            ELSE
	                // Reset to idle on invalid step
	                #step.actual := #_stepTracker.next := VacHop_Initialize_Steps#INITIAL;
	        END_CASE;

	        // Advance step when module positioned/Idle or Done and transition is enable
	        IF #enableStepTransition AND #cm_inPosition AND #mode_idleOrDone THEN
	            #step.actual := #_stepTracker.next;
	        END_IF;

	    END_IF;

	    // Manage step transitions and reset
	    #_step(forceReset := NOT #activate,
	           step := #step);
	    #_stepTracker.actual := #step.actual;

	END_REGION

	REGION Control/Equipment Modules and Modes: Commands
	    REGION Vacuum: Commands
	        CASE #step.actual OF
	            VacHop_Initialize_Steps#INITIALIZE_VACUUM:
	                // Initialize vacuum system
	                #cmd_em_vacuum := _.EM_Vac.Vac_Cmd#INITIALIZE;

	            ELSE
	                // Maintain vacuum idle
	                #cmd_em_vacuum := _.EM_Vac.Vac_Cmd#IDLE;

	        END_CASE;

	    END_REGION

	    REGION Outlet Valve: Command
	        CASE #step.actual OF
	            VacHop_Initialize_Steps#INITIALIZE_HOPPER:
	                // Initialize outlet valve
	                #cmd_em_outVlv := _.EM_outVlv.OutVlv_Cmd#INITIALIZE;

	            ELSE
	                // Maintain outlet valve idle
	                #cmd_em_outVlv := _.EM_outVlv.OutVlv_Cmd#IDLE;

	        END_CASE;

	    END_REGION

	    // Command vent mode
	    #cmd_modeVent := #step.actual = _.EM_VacHop.VacHop_Initialize_Steps#VENT;

	END_REGION

	REGION Control Modules: Commands
	    //********************************************************
	    // NA
	    //********************************************************

	END_REGION

	REGION #feedbacks
	    // Update feedback statuses
	    #feedbacks.initialized :=  #cm_inPosition AND #mode_idleOrDone AND (#step.actual = VacHop_Initialize_Steps#INITIALIZED);

	END_REGION

	REGION Status
	    // System idle when not activated system is idle when inactive
	    #status.idle := NOT #activate;

	    // System done when initialization complete
	    #status.done := NOT #status.idle AND #feedbacks.initialized;

	    // System busy during initialization sequence
	    #status.busy := NOT #status.idle AND NOT #status.done;

	END_REGION


END_FUNCTION_BLOCK
END_NAMESPACE

NAMESPACE EM_VacHop
FUNCTION_BLOCK EM_VacHop_hold
{ S7_Optimized_Access := 'TRUE' ; Published := 'TRUE' }
VERSION : 0.1
   VAR_INPUT
      enableStepTransition { ExternalAccessible := 'False'; ExternalVisible := 'False'; ExternalWritable := 'False'} : Bool := true;   // Enable Step Transition
      parameters { ExternalAccessible := 'False'; ExternalVisible := 'False'; ExternalWritable := 'False'} : VacHop_Hold_Params;   // Hold parameters
      activate { ExternalAccessible := 'False'; ExternalVisible := 'False'; ExternalWritable := 'False'} : Bool;   // Activate hold sequence
      cm_inPosition { ExternalAccessible := 'False'; ExternalVisible := 'False'; ExternalWritable := 'False'} : Bool;   // CM in position
      em_idleOrDone { ExternalAccessible := 'False'; ExternalVisible := 'False'; ExternalWritable := 'False'} : Bool;   // EM Idle or Done
      em_vacuum_idle { ExternalAccessible := 'False'; ExternalVisible := 'False'; ExternalWritable := 'False'} : Bool;   // EM Vacuum:  idle
   END_VAR

   VAR_OUTPUT
      cmd_em_vacuum { ExternalAccessible := 'False'; ExternalVisible := 'False'; ExternalWritable := 'False'} : _.EM_Vac.Vac_Cmd;   // EM_Vacuum: Command
      cmd_em_outVlv { ExternalAccessible := 'False'; ExternalVisible := 'False'; ExternalWritable := 'False'} : _.EM_OutVlv.OutVlv_Cmd;   // EM_OutVlv: Command
   END_VAR

   VAR
      status { ExternalAccessible := 'False'; ExternalVisible := 'False'; ExternalWritable := 'False'; S7_SetPoint := 'False'} : _.LIB.Util_modeStatus;   // Mode status
      feedbacks { ExternalAccessible := 'False'; ExternalVisible := 'False'; ExternalWritable := 'False'; S7_SetPoint := 'False'} : VacHop_Hold_Feedbacks;   // Feedbacks
      step { ExternalAccessible := 'False'; ExternalVisible := 'False'; ExternalWritable := 'False'; S7_SetPoint := 'False'} : _.LIB.Util_Step;   // Step status
      _step { ExternalAccessible := 'False'; ExternalVisible := 'False'; ExternalWritable := 'False'; S7_SetPoint := 'False'} : _.LIB.Step;   // Step instance
      _stepTracker { ExternalAccessible := 'False'; ExternalVisible := 'False'; ExternalWritable := 'False'} : Struct
         actual { ExternalAccessible := 'False'; ExternalVisible := 'False'; ExternalWritable := 'False'} : VacHop_Hold_Steps;   // Current step
         next { ExternalAccessible := 'False'; ExternalVisible := 'False'; ExternalWritable := 'False'} : VacHop_Hold_Steps;   // Next step
      END_STRUCT;
   END_VAR


BEGIN
	REGION Header
	    //********************************************************
	    // EM_VacHop_hold Logic
	    // Description:
	    // - Manages the hold sequence for the vacuum hopper, stopping vacuum and holding the last position of the outlet valve.
	    //********************************************************

	    REGION Revision History
	        (*
	        Author      Date        Change
	        GEA-VAR     2025-05-15  Initial version
	        *)
	    END_REGION
	END_REGION

	REGION Step
	    IF #activate THEN
	        CASE #step.actual OF
	                // Idle state, no sequence active
	            VacHop_Hold_Steps#INITIAL:
	                #_stepTracker.next := VacHop_Hold_Steps#STOP_VACUUM;

	                // Stop vacuum system
	            VacHop_Hold_Steps#STOP_VACUUM:
	                #_stepTracker.next := VacHop_Hold_Steps#HELD;

	                // Hold position
	            VacHop_Hold_Steps#HELD:
	                #_stepTracker.next := VacHop_Hold_Steps#DONE;

	                //  Hold sequence complete
	            VacHop_Hold_Steps#DONE:
	                ;

	                // Handle invalid step
	            ELSE
	                // Reset to idle on invalid step
	                #step.actual := #_stepTracker.next := VacHop_Hold_Steps#INITIAL;
	        END_CASE;

	        // Advance step when module positioned
	        IF #enableStepTransition AND #cm_inPosition AND #em_idleOrDone THEN
	            #step.actual := #_stepTracker.next;
	        END_IF;

	    END_IF;

	    // Manage step transitions and reset
	    #_step(forceReset := NOT #activate,
	           step := #step);
	    #_stepTracker.actual := #step.actual;
	END_REGION

	REGION Equipment Modules
	    REGION Vacuum: Commands
	        CASE #step.actual OF
	            VacHop_Hold_Steps#INITIAL..VacHop_Hold_Steps#STOP_VACUUM:
	                IF #em_vacuum_idle THEN
	                    #cmd_em_vacuum := _.EM_Vac.Vac_Cmd#IDLE;
	                ELSE
	                    #cmd_em_vacuum := _.EM_Vac.Vac_Cmd#STOP_VACUUM;
	                END_IF;
	            ELSE
	                #cmd_em_vacuum := _.EM_Vac.Vac_Cmd#IDLE;
	        END_CASE;

	    END_REGION

	    REGION Outlet Valve: Command
	        CASE #step.actual OF
	            VacHop_Hold_Steps#RESET_STEP:
	                #cmd_em_outVlv := _.EM_outVlv.OutVlv_Cmd#IDLE;

	            ELSE:
	                #cmd_em_outVlv := _.EM_outVlv.OutVlv_Cmd#HOLD_POSITION;

	        END_CASE;

	    END_REGION

	END_REGION

	REGION Control Modules: Commands
	    //********************************************************
	    // NA
	    //********************************************************

	END_REGION

	REGION Feedbacks
	    // Update feedback statuses
	    #feedbacks.held := #cm_inPosition AND #em_idleOrDone AND (#step.actual = VacHop_Hold_Steps#HELD) OR (#step.actual = VacHop_Hold_Steps#DONE);

	END_REGION

	REGION Status
	    // System idle when not activated
	    #status.idle := NOT #activate;

	    // System done when hold complete
	    #status.done := (NOT #status.idle) AND #cm_inPosition AND #em_idleOrDone AND (#step.actual = VacHop_Hold_Steps#DONE);

	    // System busy during hold sequence
	    #status.busy := NOT #status.idle AND NOT #status.done;

	END_REGION


END_FUNCTION_BLOCK
END_NAMESPACE

NAMESPACE EM_VacHop
FUNCTION_BLOCK EM_VacHop_purge
{ S7_Optimized_Access := 'TRUE' ; Published := 'TRUE' }
VERSION : 0.1
   VAR_INPUT
      enableStepTransition { ExternalAccessible := 'False'; ExternalVisible := 'False'; ExternalWritable := 'False'} : Bool := true;   // Enable Step Transition
      parameters { ExternalAccessible := 'False'; ExternalVisible := 'False'; ExternalWritable := 'False'} : VacHop_Purge_Params;   // Purge parameters
      activate { ExternalAccessible := 'False'; ExternalVisible := 'False'; ExternalWritable := 'False'} : Bool;   // Activate purge sequence
      cm_inPosition { ExternalAccessible := 'False'; ExternalVisible := 'False'; ExternalWritable := 'False'} : Bool;   // CM in position
      em_idleOrDone { ExternalAccessible := 'False'; ExternalVisible := 'False'; ExternalWritable := 'False'} : Bool;   // EM Idle or Done
      em_vacuum_idle { ExternalAccessible := 'False'; ExternalVisible := 'False'; ExternalWritable := 'False'} : Bool;   // EM Vacuum: Start Vacuum mode idle
      em_outVlv_outletClose { ExternalAccessible := 'False'; ExternalVisible := 'False'; ExternalWritable := 'False'} : Bool;   // EM_OutVlv: outlet valve is closed
   END_VAR

   VAR_OUTPUT
      cmd_em_vacuum { ExternalAccessible := 'False'; ExternalVisible := 'False'; ExternalWritable := 'False'} : _.EM_Vac.Vac_Cmd;   // EM_Vac command
      cmd_em_outVlv { ExternalAccessible := 'False'; ExternalVisible := 'False'; ExternalWritable := 'False'} : _.EM_OutVlv.OutVlv_Cmd;   // EM_OutVlv command
   END_VAR

   VAR
      status { ExternalAccessible := 'False'; ExternalVisible := 'False'; ExternalWritable := 'False'; S7_SetPoint := 'False'} : _.LIB.Util_modeStatus;   // Mode status
      feedbacks { ExternalAccessible := 'False'; ExternalVisible := 'False'; ExternalWritable := 'False'; S7_SetPoint := 'False'} : VacHop_Purge_Feedbacks;   // Feedbacks
      step { ExternalAccessible := 'False'; ExternalVisible := 'False'; ExternalWritable := 'False'; S7_SetPoint := 'False'} : _.LIB.Util_Step;   // Step status
      _step { ExternalAccessible := 'False'; ExternalVisible := 'False'; ExternalWritable := 'False'; S7_SetPoint := 'False'} : _.LIB.Step;   // Step instance
      _stepTracker { ExternalAccessible := 'False'; ExternalVisible := 'False'; ExternalWritable := 'False'} : Struct
         actual { ExternalAccessible := 'False'; ExternalVisible := 'False'; ExternalWritable := 'False'} : VacHop_Purge_Steps;   // Current step
         next { ExternalAccessible := 'False'; ExternalVisible := 'False'; ExternalWritable := 'False'} : VacHop_Purge_Steps;   // Next step
      END_STRUCT;
   END_VAR


BEGIN
	REGION Header
	    //********************************************************
	    // EM_VacHop_purge Logic
	    // Description:
	    // - Manages the purge sequence for the vacuum hopper by opening the outlet valve to allow a burst of purge.
	    //********************************************************

	    REGION Revision History
	        (*
	        Author      Date        Change
	        GEA-VAR     2025-05-15  Initial version
	        *)
	    END_REGION
	END_REGION

	REGION Step
	    IF #activate THEN
	        CASE #step.actual OF
	                // Idle state, no sequence active
	            VacHop_Purge_Steps#INITIAL:
	                #_stepTracker.next := VacHop_Purge_Steps#STOP_VACUUM;

	                // Stop vacuum system
	            VacHop_Purge_Steps#STOP_VACUUM:
	                #_stepTracker.next := VacHop_Purge_Steps#PURGE;

	                //  Purge hopper
	            VacHop_Purge_Steps#PURGE:
	                #_stepTracker.next := VacHop_Purge_Steps#DONE;

	                //  Purge sequence complete
	            VacHop_Purge_Steps#DONE:
	                ;

	                // Handle invalid step
	            ELSE
	                // Reset to idle on invalid step
	                #step.actual := #_stepTracker.next := VacHop_Purge_Steps#INITIAL;
	        END_CASE;

	        // Advance step when module positioned
	        IF #enableStepTransition AND #cm_inPosition AND #em_idleOrDone THEN
	            #step.actual := #_stepTracker.next;
	        END_IF;

	    END_IF;

	    // Manage step transitions and reset
	    #_step(forceReset := NOT #activate,
	           step := #step);
	    #_stepTracker.actual := #step.actual;
	END_REGION


	REGION Equipment Modules
	    REGION Vacuum: Commands
	        CASE #step.actual OF
	            VacHop_Purge_Steps#INITIAL..VacHop_Purge_Steps#STOP_VACUUM:
	                // Stop vacuum or wait for idle
	                IF #em_vacuum_idle THEN
	                    #cmd_em_vacuum := _.EM_Vac.Vac_Cmd#IDLE;
	                ELSE
	                    #cmd_em_vacuum := _.EM_Vac.Vac_Cmd#STOP_VACUUM;
	                END_IF;
	            ELSE
	                // Maintain vacuum idle
	                #cmd_em_vacuum := _.EM_Vac.Vac_Cmd#IDLE;
	        END_CASE;

	    END_REGION

	    REGION Outlet Valve: Command
	        CASE #step.actual OF
	            VacHop_Purge_Steps#INITIAL..VacHop_Purge_Steps#STOP_VACUUM:
	                // Close outlet valve or wait
	                IF NOT #em_outVlv_outletClose THEN
	                    #cmd_em_outVlv := _.EM_outVlv.OutVlv_Cmd#CLOSE_OUTLET;
	                ELSE
	                    #cmd_em_outVlv := _.EM_outVlv.OutVlv_Cmd#IDLE;

	                END_IF;

	            VacHop_Purge_Steps#PURGE:
	                // Purge outlet valve
	                #cmd_em_outVlv := _.EM_outVlv.OutVlv_Cmd#PURGE;

	            ELSE
	                // Maintain outlet valve idle
	                #cmd_em_outVlv := _.EM_outVlv.OutVlv_Cmd#IDLE;

	        END_CASE;

	    END_REGION

	END_REGION

	REGION Control Modules: Commands
	    //********************************************************
	    // NA
	    //********************************************************

	END_REGION
	//********************************************************
	// Region: #Feedback Handling
	//********************************************************
	REGION Feedbacks
	    // na

	END_REGION

	REGION Status
	    // System idle when not activated
	    #status.idle := NOT #activate;

	    // System done when purge complete
	    #status.done := (NOT #status.idle) AND #cm_inPosition AND #em_idleOrDone AND (#step.actual = VacHop_Purge_Steps#DONE);

	    // System busy during purge sequence
	    #status.busy := NOT #status.idle AND NOT #status.done;

	END_REGION


END_FUNCTION_BLOCK
END_NAMESPACE

NAMESPACE EM_VacHop
FUNCTION_BLOCK EM_VacHop_closeHopper
{ S7_Optimized_Access := 'TRUE' ; Published := 'TRUE' }
VERSION : 0.1
   VAR_INPUT
      enableStepTransition { ExternalAccessible := 'False'; ExternalVisible := 'False'; ExternalWritable := 'False'} : Bool := true;   // Enable Step Transition
      parameters { ExternalAccessible := 'False'; ExternalVisible := 'False'; ExternalWritable := 'False'} : VacHop_CloseHopper_Params;   // Close hopper parameters
      activate { ExternalAccessible := 'False'; ExternalVisible := 'False'; ExternalWritable := 'False'} : Bool;   // Activate close sequence
      cm_inPosition { ExternalAccessible := 'False'; ExternalVisible := 'False'; ExternalWritable := 'False'} : Bool;   // CM in position
      em_idleOrDone { ExternalAccessible := 'False'; ExternalVisible := 'False'; ExternalWritable := 'False'} : Bool;   // EM Idle or Done
      em_vacuum_idle { ExternalAccessible := 'False'; ExternalVisible := 'False'; ExternalWritable := 'False'} : Bool;   // EM Vacuum:  idle
      em_outVlv_outletClose { ExternalAccessible := 'False'; ExternalVisible := 'False'; ExternalWritable := 'False'} : Bool;   // EM_Hopper: outlet valve is open
   END_VAR

   VAR_OUTPUT
      cmd_em_vacuum { ExternalAccessible := 'False'; ExternalVisible := 'False'; ExternalWritable := 'False'} : _.EM_Vac.Vac_Cmd;   // EM_Vac command
      cmd_em_outVlv { ExternalAccessible := 'False'; ExternalVisible := 'False'; ExternalWritable := 'False'} : _.EM_OutVlv.OutVlv_Cmd;   // EM_OutVlv command
   END_VAR

   VAR
      status { ExternalAccessible := 'False'; ExternalVisible := 'False'; ExternalWritable := 'False'; S7_SetPoint := 'False'} : _.LIB.Util_modeStatus;   // Mode status
      feedbacks { ExternalAccessible := 'False'; ExternalVisible := 'False'; ExternalWritable := 'False'; S7_SetPoint := 'False'} : VacHop_CloseHopper_Feedbacks;   // Feedbacks
      step { ExternalAccessible := 'False'; ExternalVisible := 'False'; ExternalWritable := 'False'; S7_SetPoint := 'False'} : _.LIB.Util_Step;   // Step status
      _step { ExternalAccessible := 'False'; ExternalVisible := 'False'; ExternalWritable := 'False'; S7_SetPoint := 'False'} : _.LIB.Step;   // Step instance
      _stepTracker { ExternalAccessible := 'False'; ExternalVisible := 'False'; ExternalWritable := 'False'} : Struct
         actual { ExternalAccessible := 'False'; ExternalVisible := 'False'; ExternalWritable := 'False'} : VacHop_CloseHopper_Steps;   // Current step
         next { ExternalAccessible := 'False'; ExternalVisible := 'False'; ExternalWritable := 'False'} : VacHop_CloseHopper_Steps;   // Next step
      END_STRUCT;
   END_VAR


BEGIN
	REGION Header
	    //********************************************************
	    // EM_VacHop_closeHopper Logic
	    // Description:
	    // - Manages the hopper outlet closing sequence for the vacuum hopper, stopping vacuum and closing the outlet valve.
	    //********************************************************

	    REGION Revision History
	        (*
	        Author      Date        Change
	        GEA-VAR     2025-05-15  Initial version
	        *)
	    END_REGION
	END_REGION

	REGION Step
	    IF #activate THEN
	        CASE #step.actual OF
	                // Idle state, no sequence active
	            VacHop_CloseHopper_Steps#INITIAL:
	                #_stepTracker.next := VacHop_CloseHopper_Steps#STOP_VACUUM;

	                // Stop vacuum system
	            VacHop_CloseHopper_Steps#STOP_VACUUM:
	                #_stepTracker.next := VacHop_CloseHopper_Steps#CLOSE_OUTLET;

	                //  Close outlet valve
	            VacHop_CloseHopper_Steps#CLOSE_OUTLET:
	                #_stepTracker.next := VacHop_CloseHopper_Steps#DONE;

	                //  Outlet valve closed, sequence complete
	            VacHop_CloseHopper_Steps#DONE:
	                ;

	                // Handle invalid step
	            ELSE
	                // Reset to idle on invalid step
	                #step.actual := #_stepTracker.next := VacHop_CloseHopper_Steps#INITIAL;
	        END_CASE;

	        // Advance step when module positioned
	        IF #enableStepTransition AND #cm_inPosition AND #em_idleOrDone THEN
	            #step.actual := #_stepTracker.next;
	        END_IF;

	    END_IF;

	    // Manage step transitions and reset
	    #_step(forceReset := NOT #activate,
	           step := #step);
	    #_stepTracker.actual := #step.actual;
	END_REGION

	REGION Control/Equipment Modules and Modes: Commands

	    REGION Vacuum: Commands
	        CASE #step.actual OF
	            VacHop_CloseHopper_Steps#INITIAL..VacHop_CloseHopper_Steps#STOP_VACUUM:
	                // Stop vacuum or wait for idle
	                IF #em_vacuum_idle THEN
	                    #cmd_em_vacuum := _.EM_Vac.Vac_Cmd#IDLE;
	                ELSE
	                    #cmd_em_vacuum := _.EM_Vac.Vac_Cmd#STOP_VACUUM;
	                END_IF;
	            ELSE
	                #cmd_em_vacuum := _.EM_Vac.Vac_Cmd#IDLE;
	        END_CASE;

	    END_REGION

	    REGION Outlet Valve: Command
	        CASE #step.actual OF
	            VacHop_CloseHopper_Steps#INITIAL..VacHop_CloseHopper_Steps#STOP_VACUUM:
	                IF NOT #em_outVlv_outletClose THEN
	                    #cmd_em_outVlv := _.EM_outVlv.OutVlv_Cmd#OPEN_OUTLET;
	                ELSE
	                    #cmd_em_outVlv := _.EM_outVlv.OutVlv_Cmd#IDLE;
	                END_IF;
	            VacHop_CloseHopper_Steps#CLOSE_OUTLET:
	                IF NOT #em_outVlv_outletClose THEN
	                    #cmd_em_outVlv := _.EM_outVlv.OutVlv_Cmd#CLOSE_OUTLET;
	                ELSE
	                    #cmd_em_outVlv := _.EM_outVlv.OutVlv_Cmd#IDLE;
	                END_IF;
	            ELSE
	                // Maintain outlet valve closed
	                #cmd_em_outVlv := _.EM_outVlv.OutVlv_Cmd#IDLE;
	        END_CASE;

	    END_REGION

	END_REGION

	REGION Control Modules: Commands
	    //********************************************************
	    // NA
	    //********************************************************

	END_REGION

	REGION Feedbacks
	    // NA

	END_REGION

	REGION Status
	    // System idle when not activated
	    #status.idle := NOT #activate;

	    // System done when hopper closed
	    #status.done := (NOT #status.idle) AND #cm_inPosition AND #em_idleOrDone AND (#step.actual = VacHop_CloseHopper_Steps#DONE);

	    // System busy during close sequence
	    #status.busy := NOT #status.idle AND NOT #status.done;

	END_REGION


END_FUNCTION_BLOCK
END_NAMESPACE

NAMESPACE EM_Vac
FUNCTION_BLOCK EM_Vac
{ S7_Optimized_Access := 'TRUE' ; Published := 'TRUE' }
VERSION : 0.1
   VAR_INPUT
      enableStepTransition { ExternalAccessible := 'False'; ExternalVisible := 'False'; ExternalWritable := 'False'} : Bool := True;   // Enable step transition
      vacuumInputs { ExternalAccessible := 'False'; ExternalVisible := 'False'; ExternalWritable := 'False'} : Vac_inputs;   // EM inputs
      emptyLine { ExternalAccessible := 'False'; ExternalVisible := 'False'; ExternalWritable := 'False'} : Bool;   // Request empty line
   END_VAR

   VAR_OUTPUT
      cm_inPosition { ExternalAccessible := 'False'; ExternalVisible := 'False'; ExternalWritable := 'False'} : Bool;   // CM in position
      cmd_isolationVlvOpen { ExternalAccessible := 'False'; ExternalVisible := 'False'; ExternalWritable := 'False'} : Bool;   // Command to open isolation valve
      cmd_vacuumVlvOpen { ExternalAccessible := 'False'; ExternalVisible := 'False'; ExternalWritable := 'False'} : Bool;   // Command to open vacuum valve
      setpoint_vacuumControlVlv { ExternalAccessible := 'False'; ExternalVisible := 'False'; ExternalWritable := 'False'} : Real;   // Vacuum control valve setpoint
   END_VAR

   VAR
      interface { ExternalAccessible := 'False'; ExternalVisible := 'False'; ExternalWritable := 'False'; S7_SetPoint := 'False'} : Vac_interface;
      parameters : Vac_parameters;
      _initialize { ExternalAccessible := 'False'; ExternalVisible := 'False'; ExternalWritable := 'False'; S7_SetPoint := 'False'} : EM_Vac_initialize;
      _startVacuum { ExternalAccessible := 'False'; ExternalVisible := 'False'; ExternalWritable := 'False'; S7_SetPoint := 'False'} : EM_Vac_startVacuum;
      _stopVacuum { ExternalAccessible := 'False'; ExternalVisible := 'False'; ExternalWritable := 'False'; S7_SetPoint := 'False'} : EM_Vac_stopVacuum;
      _outputs { ExternalAccessible := 'False'; ExternalVisible := 'False'; ExternalWritable := 'False'} : Struct
         cmd_isolationVlvOpen { ExternalAccessible := 'False'; ExternalVisible := 'False'; ExternalWritable := 'False'} : Bool;
         cmd_vacuumVlvOpen { ExternalAccessible := 'False'; ExternalVisible := 'False'; ExternalWritable := 'False'} : Bool;
      END_STRUCT;
   END_VAR

   VAR_TEMP
      temp_modes_idle_or_done : Bool;   // excluding "Initialize mode"
   END_VAR


BEGIN
	REGION Header
	    //********************************************************
	    // EM_Vac Logic
	    // Description:
	    // - Main controller for the vacuum system, managing initialization, start, and stop sequences.
	    //********************************************************

	    REGION Revision History
	        (*
	            Author      Date        Change
	            GEA-VAR     15MAY25     Initial version
	        *)
	    END_REGION

	END_REGION

	REGION Check CM/EM(mode) in position
	    // Set control module position status
	    #cm_inPosition :=
	        ((#_outputs.cmd_isolationVlvOpen AND #vacuumInputs.isolationVlv_isOpen) OR ((NOT #_outputs.cmd_isolationVlvOpen) AND #vacuumInputs.isolationVlv_isClosed)) AND
	        ((#_outputs.cmd_vacuumVlvOpen AND #vacuumInputs.vacuumVlv_isOpen) OR ((NOT #_outputs.cmd_vacuumVlvOpen) AND #vacuumInputs.vacuumVlv_isClosed));

	    // Check if modes are idle or done
	    #temp_modes_idle_or_done :=
	        (#_startVacuum.status.idle OR #_startVacuum.status.done) AND
	        (#_stopVacuum.status.idle OR #_stopVacuum.status.done);

	END_REGION

	REGION Initialize
	    // Run initialization sequence
	    #_initialize(en_stepTrans:=#enableStepTransition,
	                 activate:=(#interface.cmd = Vac_Cmd#INITIALIZE),
	                 cm_inPosition:=#cm_inPosition,
	                 mode_idleOrDone:=#temp_modes_idle_or_done);

	END_REGION

	REGION Start Vacuum
	    // Configure parameters for start sequence
	    REGION Parameters
	        #_startVacuum.parameters.minVacuumAirFlow := #parameters.fixed.vacuumMinAirFlow;
	        #_startVacuum.parameters.vacuumBuildUpTimer := #parameters.fixed.vacuumBuildUpTimer;
	        #_startVacuum.parameters.vacuumControlSP := #parameters.fixed.vacuumControlSP;
	        #_startVacuum.parameters.vacuumControlMinOpening := #parameters.fixed.vacuumControlMinOpening;
	        #_startVacuum.parameters.minTimeLineEmpty := #parameters.variable.minTimeLineEmpty;
	    END_REGION

	    // Activate start sequence on command
	    #_startVacuum(enableStepTransition:=#enableStepTransition,
	                  activate := (#interface.cmd = Vac_Cmd#START_VACUUM) OR #_initialize.cmd_modeStartVacuum,
	                  emptyLine:=#emptyLine,
	                  cm_inPosition:=#cm_inPosition,
	                  AHU_minAirflowReached := #vacuumInputs.AHU_minAirflowReached,
	                  vacuumAirflow_PV := #vacuumInputs.vacuumAirflow_PV);
	END_REGION

	REGION Stop Vacuum
	    // Configure parameters for stop sequence
	    REGION Parameters
	        #_stopVacuum.parameters.isolationVlvCloseDelay := #parameters.variable.isolationVlvCloseDelay;
	        #_stopVacuum.parameters.vacuumVlvCloseDelay := #parameters.fixed.vacuumVlvCloseDelay;
	        #_stopVacuum.parameters.vacuumControlSP := #parameters.fixed.vacuumControlSP;
	        #_stopVacuum.parameters.vacuumControlMinOpening := #parameters.fixed.vacuumControlMinOpening;

	    END_REGION

	    // Activate stop sequence on command
	    #_stopVacuum(enableStepTransition:=#enableStepTransition,
	                 activate := (#interface.cmd = Vac_Cmd#STOP_VACUUM) OR #_initialize.cmd_modeStopVacuum,
	                 cm_inPosition:=#cm_inPosition,
	                 vacuumVlv_isOpen := #vacuumInputs.vacuumVlv_isOpen,
	                 vacuumVlv_isClosed := #vacuumInputs.vacuumVlv_isClosed,
	                 isolationVlv_isOpen := #vacuumInputs.isolationVlv_isOpen,
	                 isolationVlv_isClosed := #vacuumInputs.isolationVlv_isClosed);

	END_REGION

	REGION Outputs
	    // Aggregate valve commands
	    #cmd_isolationVlvOpen := #_outputs.cmd_isolationVlvOpen := #_startVacuum.cmd_isolationVlvOpen OR #_stopVacuum.cmd_isolationVlvOpen;
	    #cmd_vacuumVlvOpen := #_outputs.cmd_vacuumVlvOpen := #_startVacuum.cmd_vacuumVlvOpen OR #_stopVacuum.cmd_vacuumVlvOpen;

	    // Select maximum setpoint for valve
	    #setpoint_vacuumControlVlv := MAX_REAL(IN1 := #_startVacuum.setpoint_vacuumControlVlv, IN2 := #_stopVacuum.setpoint_vacuumControlVlv);

	END_REGION

	REGION Feedbacks
	    #interface.feedbacks.isolationVlvOpen := (NOT #_startVacuum.status.idle) AND #vacuumInputs.isolationVlv_isOpen;
	    // Update mode feedbacks
	    REGION Modes
	        #interface.feedbacks.modes.initialize := #_initialize.feedbacks;
	        #interface.feedbacks.modes.startVacuum := #_startVacuum.feedbacks;
	        #interface.feedbacks.modes.stopVacuum := #_stopVacuum.feedbacks;
	    END_REGION

	END_REGION

	REGION Check CM/EM(mode) in position
	    // Set control module position status
	    #cm_inPosition :=
	    ((#_outputs.cmd_isolationVlvOpen AND #vacuumInputs.isolationVlv_isOpen) OR ((NOT #_outputs.cmd_isolationVlvOpen) AND #vacuumInputs.isolationVlv_isClosed)) AND
	    ((#_outputs.cmd_vacuumVlvOpen AND #vacuumInputs.vacuumVlv_isOpen) OR ((NOT #_outputs.cmd_vacuumVlvOpen) AND #vacuumInputs.vacuumVlv_isClosed));

	    // Check if modes are idle or done
	    #temp_modes_idle_or_done := (#_startVacuum.status.idle OR #_startVacuum.status.done) AND (#_stopVacuum.status.idle OR #_stopVacuum.status.done);


	END_REGION

	REGION Status
	    // Set overall and mode statuses
	    #interface.status.done := #_initialize.status.done OR
	        ((NOT #_initialize.status.busy) AND (#_startVacuum.status.done OR #_stopVacuum.status.done));
	    #interface.status.busy := #_initialize.status.busy OR #_startVacuum.status.busy OR #_stopVacuum.status.busy OR (#interface.status.busy AND (NOT #cm_inPosition));
	    #interface.status.idle := (NOT (#interface.status.busy OR #interface.status.done)) AND #cm_inPosition AND #temp_modes_idle_or_done AND #_initialize.status.idle;
	    #interface.status.stopAlmActive := _.EM.TODO.alm;
	    #interface.status.abortAlmActive := _.EM.TODO.alm;

	    // Modes
	    #interface.modesStatus.initialize := #_initialize.status;
	    #interface.modesStatus.startVacuum := #_startVacuum.status;
	    #interface.modesStatus.stopVacuum := #_stopVacuum.status;

	END_REGION

END_FUNCTION_BLOCK
END_NAMESPACE

NAMESPACE EM_VacHop
FUNCTION_BLOCK EM_VacHop
{ S7_Optimized_Access := 'TRUE' ; Published := 'TRUE' }
VERSION : 0.1
   VAR_INPUT
      enableStepTransition { ExternalAccessible := 'False'; ExternalVisible := 'False'; ExternalWritable := 'False'} : Bool := True;   // Enable step transition
      vacHopInputs { ExternalAccessible := 'False'; ExternalVisible := 'False'; ExternalWritable := 'False'} : VacHop_inputs;   // EM inputs
      emptyLine { ExternalAccessible := 'False'; ExternalVisible := 'False'; ExternalWritable := 'False'} : Bool;   // Request empty line
   END_VAR

   VAR_OUTPUT
      cm_inPosition { ExternalAccessible := 'False'; ExternalVisible := 'False'; ExternalWritable := 'False'} : Bool;
      cmd_isolationVlvOpen { ExternalAccessible := 'False'; ExternalVisible := 'False'; ExternalWritable := 'False'} : Bool;
      cmd_vacuumVlvOpen { ExternalAccessible := 'False'; ExternalVisible := 'False'; ExternalWritable := 'False'} : Bool;
      cmd_vacuumControlVlvOpen { ExternalAccessible := 'False'; ExternalVisible := 'False'; ExternalWritable := 'False'} : Bool;
      setpoint_vacuumControlVlv { ExternalAccessible := 'False'; ExternalVisible := 'False'; ExternalWritable := 'False'} : Real;
      cmd_outletVlvOpen { ExternalAccessible := 'False'; ExternalVisible := 'False'; ExternalWritable := 'False'} : Bool;
      cmd_ventVlvOpen { ExternalAccessible := 'False'; ExternalVisible := 'False'; ExternalWritable := 'False'} : Bool;
   END_VAR

   VAR
      interface { ExternalAccessible := 'False'; ExternalVisible := 'False'; ExternalWritable := 'False'; S7_SetPoint := 'False'} : VacHop_interface;
      parameters : VacHop_parameters;
      _em_vacuum { ExternalAccessible := 'False'; ExternalVisible := 'False'; ExternalWritable := 'False'; S7_SetPoint := 'False'} : _.EM_Vac.EM_Vac;   // EM Vacuum instance
      _em_outVlv { ExternalAccessible := 'False'; ExternalVisible := 'False'; ExternalWritable := 'False'; S7_SetPoint := 'False'} : _.EM_OutVlv.EM_OutVlv;   // EM Hopper instance
      _initialize { ExternalAccessible := 'False'; ExternalVisible := 'False'; ExternalWritable := 'False'; S7_SetPoint := 'False'} : EM_VacHop_initialize;
      _discharge { ExternalAccessible := 'False'; ExternalVisible := 'False'; ExternalWritable := 'False'; S7_SetPoint := 'False'} : EM_VacHop_discharge;
      _vent { ExternalAccessible := 'False'; ExternalVisible := 'False'; ExternalWritable := 'False'; S7_SetPoint := 'False'} : EM_VacHop_vent;
      _openHopper { ExternalAccessible := 'False'; ExternalVisible := 'False'; ExternalWritable := 'False'; S7_SetPoint := 'False'} : EM_VacHop_openHopper;
      _evacuate { ExternalAccessible := 'False'; ExternalVisible := 'False'; ExternalWritable := 'False'; S7_SetPoint := 'False'} : EM_VacHop_evacuate;
      _flowThrough { ExternalAccessible := 'False'; ExternalVisible := 'False'; ExternalWritable := 'False'; S7_SetPoint := 'False'} : EM_VacHop_flowThrough;
      _purge { ExternalAccessible := 'False'; ExternalVisible := 'False'; ExternalWritable := 'False'; S7_SetPoint := 'False'} : EM_VacHop_purge;
      _closeHopper { ExternalAccessible := 'False'; ExternalVisible := 'False'; ExternalWritable := 'False'; S7_SetPoint := 'False'} : EM_VacHop_closeHopper;
      _hold { ExternalAccessible := 'False'; ExternalVisible := 'False'; ExternalWritable := 'False'} : EM_VacHop_hold;
      _outputs { ExternalAccessible := 'False'; ExternalVisible := 'False'; ExternalWritable := 'False'} : Struct
         cmd_ventVlvOpen { ExternalAccessible := 'False'; ExternalVisible := 'False'; ExternalWritable := 'False'} : Bool;
      END_STRUCT;
   END_VAR

   VAR_TEMP
      temp_em_idle_or_done : Bool;
   END_VAR


BEGIN
	REGION Header
	    //********************************************************
	    // EM_VacHop Logic
	    // Description: Handles the Vacuum Hopper initialization process. The initialize block is activated
	    //********************************************************

	    REGION Revision History
	        (*
	            Author      Date        Change
	            GEA-VAR     15MAY25     Initial version
	        *)
	    END_REGION

	END_REGION

	REGION Check CM/EM(mode) in position
	    // Set control module position status
	    #cm_inPosition :=
	        #_em_vacuum.cm_inPosition AND #_em_outVlv.cm_inPosition AND
	        ((#_outputs.cmd_ventVlvOpen AND #vacHopInputs.ventVlv_isOpen) OR ((NOT #_outputs.cmd_ventVlvOpen) AND #vacHopInputs.ventVlv_isClosed));

	    // Check if modes are idle or done
	    #temp_em_idle_or_done :=
	        (#_em_vacuum.interface.status.idle OR #_em_vacuum.interface.status.done) AND
	        (#_em_outVlv.interface.status.idle OR #_em_outVlv.interface.status.done);

	END_REGION

	REGION Initialize
	    #_initialize(enableStepTransition:=#enableStepTransition,
	                 activate:=(#interface.cmd = VacHop_Cmd#INITIALIZE),
	                 cm_inPosition:=#cm_inPosition,
	                 mode_idleOrDone:=#temp_em_idle_or_done);

	END_REGION

	REGION Discharge
	    REGION Parameters
	        #_discharge.parameters.na := FALSE;

	    END_REGION

	    #_discharge(enableStepTransition:=#enableStepTransition,
	                activate:=(#interface.cmd = VacHop_Cmd#DISCHARGE),
	                cm_inPosition:=#cm_inPosition,
	                em_idleOrDone:=#temp_em_idle_or_done,
	                em_vacuum_idle:=#_em_vacuum.interface.status.idle,
	                em_outVlv_outletClose:=#vacHopInputs.em_outVlv_inputs.outletVlv_isClosed);

	END_REGION

	REGION Vent
	    REGION Parameters
	        #_vent.parameters.ventTime := #parameters.fixed.ventTime;

	    END_REGION

	    #_vent(enableStepTransition:=#enableStepTransition,
	           activate:=(#interface.cmd = VacHop_Cmd#VENT) OR #_initialize.cmd_modeVent,
	           cm_inPosition:=#cm_inPosition,
	           em_idleOrDone:=#temp_em_idle_or_done,
	           em_vacuum_idle:=#_em_vacuum.interface.status.idle,
	           em_outVlv_outletClose:=#vacHopInputs.em_outVlv_inputs.outletVlv_isClosed);

	END_REGION

	REGION Open Hopper
	    REGION Parameters
	        #_openHopper.parameters.na := FALSE;

	    END_REGION

	    #_openHopper(enableStepTransition:=#enableStepTransition,
	                 activate := (#interface.cmd = VacHop_Cmd#OPEN_HOPPER),
	                 cm_inPosition:=#cm_inPosition,
	                 em_idleOrDone:=#temp_em_idle_or_done,
	                 em_vacuum_idle:=#_em_vacuum.interface.status.idle,
	                 em_outVlv_outletClose := #vacHopInputs.em_outVlv_inputs.outletVlv_isClosed);

	END_REGION

	REGION Evacuate
	    REGION Parameters
	        #_evacuate.parameters.na := FALSE;

	    END_REGION

	    #_evacuate(enableStepTransition:=#enableStepTransition,
	               activate := (#interface.cmd = VacHop_Cmd#EVACUATE),
	               cm_inPosition:=#cm_inPosition,
	               em_idleOrDone:=#temp_em_idle_or_done,
	               em_vacuum_startVacuum_idle:=#_em_vacuum.interface.modesStatus.startVacuum.idle,
	               em_outVlv_outletClose := #vacHopInputs.em_outVlv_inputs.outletVlv_isClosed);

	END_REGION

	REGION Flowthrough
	    REGION Parameters
	        #_flowThrough.parameters.na := FALSE;

	    END_REGION

	    // Activate stop logic when STOP_VACUUM command is issued or initialize requires it
	    #_flowThrough(activate := (#interface.cmd = VacHop_Cmd#FLOWTHROUGHT),
	                  cm_inPosition:=#cm_inPosition,
	                  em_idleOrDone:=#temp_em_idle_or_done,
	                  em_vacuum_startVacuum_idle:=#_em_vacuum.interface.modesStatus.startVacuum.idle,
	                  em_outVlv_outletClose := #vacHopInputs.em_outVlv_inputs.outletVlv_isClosed);

	END_REGION

	REGION Purge
	    REGION Parameters
	        #_purge.parameters.na := FALSE;

	    END_REGION

	    #_purge(enableStepTransition:=#enableStepTransition,
	            activate := (#interface.cmd = VacHop_Cmd#PURGE),
	            cm_inPosition:=#cm_inPosition,
	            em_idleOrDone:=#temp_em_idle_or_done,
	            em_vacuum_idle:=#_em_vacuum.interface.status.idle,
	            em_outVlv_outletClose := #vacHopInputs.em_outVlv_inputs.outletVlv_isClosed);
	END_REGION

	REGION Close Hopper
	    REGION Parameters
	        #_closeHopper.parameters.na := FALSE;

	    END_REGION

	    #_closeHopper(enableStepTransition:=#enableStepTransition,
	                  activate := (#interface.cmd = VacHop_Cmd#CLOSE_HOPPER),
	                  cm_inPosition := #cm_inPosition,
	                  em_idleOrDone := #temp_em_idle_or_done,
	                  em_vacuum_idle := #_em_vacuum.interface.status.idle,
	                  em_outVlv_outletClose := #vacHopInputs.em_outVlv_inputs.outletVlv_isClosed);

	END_REGION

	REGION Hold
	    REGION Parameters
	        #_hold.parameters.na := FALSE;

	    END_REGION

	    #_hold(enableStepTransition:=#enableStepTransition,
	           activate := (#interface.cmd = VacHop_Cmd#HOLD),
	           cm_inPosition := #cm_inPosition,
	           em_idleOrDone := #temp_em_idle_or_done,
	           em_vacuum_idle := #_em_vacuum.interface.status.idle);

	END_REGION


	//********************************************************
	// Region: Command Mapping
	//********************************************************
	REGION Commands
	    REGION Equipment Modules
	        REGION Vacuum
	            REGION Parameters
	                // Fixed
	                #_em_vacuum.parameters.fixed := #parameters.fixed.em_vac;

	                // Variable
	                #_em_vacuum.parameters.variable.isolationVlvCloseDelay := #parameters.fixed.isolationVlvCloseDelay;
	                #_em_vacuum.parameters.variable.minTimeLineEmpty := #parameters.variable.transferLineEmptyTime;

	            END_REGION


	            REGION Control/Command
	                #_em_vacuum.interface.cmd := MAX_USINT(IN1 := #_initialize.cmd_em_vacuum,
	                                                       IN2 := #_discharge.cmd_em_vacuum,
	                                                       IN3 := #_vent.cmd_em_vacuum,
	                                                       IN4 := #_openHopper.cmd_em_vacuum,
	                                                       IN5 := #_evacuate.cmd_em_vacuum,
	                                                       IN6 := #_flowThrough.cmd_em_vacuum,
	                                                       IN7 := #_purge.cmd_em_vacuum,
	                                                       IN8 := #_closeHopper.cmd_em_vacuum,
	                                                       IN9 := #_hold.cmd_em_vacuum);
	            END_REGION

	            #_em_vacuum(enableStepTransition:=#enableStepTransition,
	                        vacuumInputs:=#vacHopInputs.em_vac_inputs,
	                        emptyLine:=#emptyLine,
	                        cmd_isolationVlvOpen=>#cmd_isolationVlvOpen,
	                        cmd_vacuumVlvOpen=>#cmd_vacuumVlvOpen,
	                        setpoint_vacuumControlVlv=>#setpoint_vacuumControlVlv);

	        END_REGION

	        REGION Hopper
	            REGION Parameters
	                // Fixed
	                #_em_outVlv.parameters.fixed := #parameters.fixed.em_outVlv;

	                // Variable
	                #_em_outVlv.parameters.variable.dischargeTime := #parameters.fixed.dischargeTime;

	            END_REGION

	            REGION Control/Command
	                #_em_outVlv.interface.cmd := MAX_USINT(IN1 := #_initialize.cmd_em_outVlv,
	                                                       IN2 := #_discharge.cmd_em_outVlv,
	                                                       IN3 := #_vent.cmd_em_outVlv,
	                                                       IN4 := #_openHopper.cmd_em_outVlv,
	                                                       IN5 := #_evacuate.cmd_em_outVlv,
	                                                       IN6 := #_flowThrough.cmd_em_outVlv,
	                                                       IN7 := #_purge.cmd_em_outVlv,
	                                                       IN8 := #_closeHopper.cmd_em_outVlv,
	                                                       IN9 := #_hold.cmd_em_outVlv);
	            END_REGION

	            #_em_outVlv(enableStepTransition:=#enableStepTransition,
	                        outletValveInputs:=#vacHopInputs.em_outVlv_inputs,
	                        cmd_outletVlvOpen=>#cmd_outletVlvOpen);

	        END_REGION

	    END_REGION

	    REGION Control Modules
	        #cmd_ventVlvOpen := #_outputs.cmd_ventVlvOpen := #_vent.cmd_ventVlvOpen;

	    END_REGION
	END_REGION


	REGION Feedbacks
	    #interface.feedbacks.transferLineEmpty := #interface.feedbacks.em_vacuum.modes.startVacuum.minTimeLineEmptyReached;

	    REGION Modes
	        #interface.feedbacks.modes.initialize := #_initialize.feedbacks;
	        #interface.feedbacks.modes.discharge := #_discharge.feedbacks;
	        #interface.feedbacks.modes.vent := #_vent.feedbacks;
	        #interface.feedbacks.modes.openHopper := #_openHopper.feedbacks;
	        #interface.feedbacks.modes.evacuate := #_evacuate.feedbacks;
	        #interface.feedbacks.modes.flowThrough := #_flowThrough.feedbacks;
	        #interface.feedbacks.modes.purge := #_purge.feedbacks;
	        #interface.feedbacks.modes.closeHopper := #_closeHopper.feedbacks;
	        #interface.feedbacks.modes.hold := #_hold.feedbacks;

	    END_REGION

	    REGION Equipment Modules
	        #interface.feedbacks.em_vacuum := #_em_vacuum.interface.feedbacks;
	        #interface.feedbacks.em_hopper := #_em_outVlv.interface.feedbacks;

	    END_REGION


	END_REGION


	REGION Check CM/EM(mode) in position
	    // Set control module position status
	    #cm_inPosition := #_em_vacuum.cm_inPosition AND #_em_outVlv.cm_inPosition AND
	        ((#_outputs.cmd_ventVlvOpen AND #vacHopInputs.ventVlv_isOpen) OR ((NOT #_outputs.cmd_ventVlvOpen) AND #vacHopInputs.ventVlv_isClosed));

	    // Check if modes are idle or done
	    #temp_em_idle_or_done :=
	        (#_em_vacuum.interface.status.idle OR #_em_vacuum.interface.status.done) AND
	        (#_em_outVlv.interface.status.idle OR #_em_outVlv.interface.status.done);

	END_REGION

	REGION Status
	    #interface.status.done :=
	        #_initialize.status.done OR #_discharge.status.done OR #_openHopper.status.done OR #_evacuate.status.done OR #_flowThrough.status.done OR #_purge.status.done OR #_closeHopper.status.done OR #_hold.status.done OR
	        ((NOT #_initialize.status.busy) AND #_vent.status.done);
	    #interface.status.busy :=
	        #_initialize.status.busy OR #_discharge.status.busy OR #_vent.status.busy OR #_openHopper.status.busy OR #_evacuate.status.busy OR #_flowThrough.status.busy OR #_purge.status.busy OR #_closeHopper.status.busy OR #_hold.status.busy;
	    #interface.status.idle := NOT (#interface.status.busy OR #interface.status.done);
	    #interface.status.stopAlmActive := _.EM.TODO.alm;
	    #interface.status.abortAlmActive := _.EM.TODO.alm;

	    // Modes
	    #interface.modesStatus.initialize := #_initialize.status;
	    #interface.modesStatus.discharge := #_discharge.status;
	    #interface.modesStatus.vent := #_vent.status;
	    #interface.modesStatus.openHopper := #_openHopper.status;
	    #interface.modesStatus.evacuate := #_evacuate.status;
	    #interface.modesStatus.flowThrough := #_flowThrough.status;
	    #interface.modesStatus.purge := #_purge.status;
	    #interface.modesStatus.closeHopper := #_closeHopper.status;
	    #interface.modesStatus.hold := #_hold.status;

	END_REGION

END_FUNCTION_BLOCK
END_NAMESPACE

